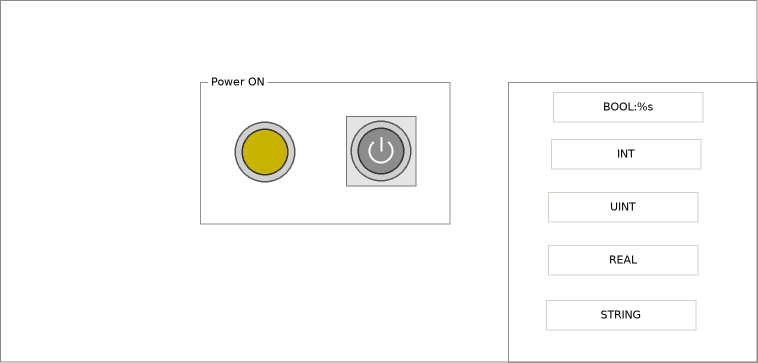
VISUALIZATION HMI  // 758x363
    GroupBox (200,74 250x150), "Power ON"
        Lamp1 (30,43 70x70), variable: MAIN.bEnable, style: Lamp-Lamp1-Yellow
        PowerSwitch (146,42 70x70), variable: MAIN.bStart, behaviour: TOGGLE, style: Switch-PowerSwitch-Gray
    GroupBox (508,74 250x289)
        Textfield (45,18 150x30), "BOOL:%s", text variable: MAIN.bEnable
        Textfield (43,65 150x30), "INT"
        Textfield (40,118 150x30), "UINT"
        Textfield (40,171 150x30), "REAL"
        Textfield (38,226 150x30), "STRING"
END_VISUALIZATION

(* stored: Version 1.1.0.1, ProductVersion 3.1.4024.12
   Visu HMI: Id {c37f6f2b-1c97-4e24-8c98-b4f32a8fe82b} *)
